FUNCTION_BLOCK FB_Event IMPLEMENTS I_Event
VAR_INPUT
END_VAR
VAR_OUTPUT
END_VAR
VAR
	iHandler:			I_Handler;
	stDebug:			ST_Event;
	stInfo:				ST_Event;
	stWarning:			ST_Event;
	stError:			ST_Event;
END_VAR

IF stDebug.bActive THEN
	stDebug.bActive:= FALSE;
ELSE
	stDebug.nTimestamp:= 0;
END_IF

IF stInfo.bActive THEN
	stInfo.bActive:= FALSE;	
ELSE
	stInfo.nTimestamp:= 0;		
END_IF

IF stWarning.bActive THEN
	stWarning.bActive:= FALSE;	
ELSE
	stWarning.nTimestamp:= 0;	
END_IF

IF stError.bActive THEN
	stError.bActive:= FALSE;	
ELSE
	stError.nTimestamp:= 0;	
END_IF

METHOD PUBLIC M_Debug
VAR_INPUT
	sMessage:	STRING(255);
	nID:		DINT;
END_VAR
stDebug.bActive:= TRUE;
stDebug.bEvent:= FALSE;
IF stDebug.sMessage <> sMessage THEN
	stDebug.bEvent:= TRUE;
END_IF
IF stDebug.nTimestamp = 0 THEN
	stDebug.nTimestamp:= F_GetSystemTime();
	stDebug.bEvent:= TRUE;
END_IF
stDebug.eEvent:= E_Event.Debug;
stDebug.sMessage:= sMessage;
stDebug.nID:= nID;

IF iHandler <> 0 THEN
	iHandler.M_Request(stDebug);
END_IF
END_METHOD

METHOD PUBLIC M_Error
VAR_INPUT
	sMessage:	STRING(255);
	nID:		DINT;
END_VAR
stError.bActive:= TRUE;
stError.bEvent:= FALSE;
IF stError.sMessage <> sMessage THEN
	stError.bEvent:= TRUE;
END_IF
IF stError.nTimestamp = 0 THEN
	stError.nTimestamp:= F_GetSystemTime();
	stError.bEvent:= TRUE;
END_IF
stError.eEvent:= E_Event.Error;
stError.sMessage:= sMessage;
stError.nID:= nID;

IF iHandler <> 0 THEN
	iHandler.M_Request(stError);
END_IF
END_METHOD

METHOD PUBLIC M_Info
VAR_INPUT
	sMessage:	STRING(255);
	nID:		DINT;
END_VAR
stInfo.bActive:= TRUE;
stInfo.bEvent:= FALSE;
IF stInfo.sMessage <> sMessage THEN
	stInfo.bEvent:= TRUE;
END_IF
IF stInfo.nTimestamp = 0 THEN
	stInfo.nTimestamp:= F_GetSystemTime();
	stInfo.bEvent:= TRUE;
END_IF
stInfo.eEvent:= E_Event.Info;
stInfo.sMessage:= sMessage;
stInfo.nID:= nID;

IF iHandler <> 0 THEN
	iHandler.M_Request(stInfo);
END_IF
END_METHOD

METHOD M_Warning
VAR_INPUT
	sMessage:	STRING(255);
	nID:		DINT;
END_VAR
stWarning.bActive:= TRUE;
stWarning.bEvent:= FALSE;
IF stWarning.sMessage <> sMessage THEN
	stWarning.bEvent:= TRUE;
END_IF
IF stWarning.nTimestamp = 0 THEN
	stWarning.nTimestamp:= F_GetSystemTime();
	stWarning.bEvent:= TRUE;
END_IF
stWarning.eEvent:= E_Event.Warning;
stWarning.sMessage:= sMessage;
stWarning.nID:= nID;

IF iHandler <> 0 THEN
	iHandler.M_Request(stWarning);
END_IF
END_METHOD

PROPERTY PUBLIC P_Handler : I_Handler
GET
P_Handler:= iHandler;
END_GET
SET
iHandler:= P_Handler;
END_SET
END_PROPERTY

END_FUNCTION_BLOCK

(* stored: Version 1.1.0.1, ProductVersion 3.1.4024.12
   POU FB_Event: Id {1dcb84ec-d695-4d6f-a3ff-99e012891880}, SpecialFunc None
   Method M_Debug: Id {51e168c5-af65-4a41-9856-1decc56cb137}
   Method M_Error: Id {5d080c91-569f-424a-821e-4296fce43891}
   Method M_Info: Id {d7d83d14-1059-441b-8e79-b513a6fba4c9}
   Method M_Warning: Id {da4a05a4-d352-4379-97c7-69430f6a9b91}
   Property P_Handler: Id {47eda2e3-f16a-4044-b37b-35367509189b}
   Get Get: Id {539e947b-f005-4d1f-9833-5c2b5c69a723}
   Set Set: Id {76fd1b75-9a5b-43f6-8e2f-6b1bcc67aaf5} *)
